// TIA Portal V16 export
// export: Created 2022-09-01T13:58:56.9257321Z, ExportSetting WithDefaults, DisplayName Totally Integrated Automation Portal, DisplayVersion V16, DisplayName TIA Portal Version Control Interface, DisplayVersion V16, DisplayName TIA Portal Openness, DisplayVersion V16, DisplayName STEP 7 Professional, DisplayVersion V16, DisplayName STEP 7 Safety, DisplayVersion V16, DisplayName WinCC Advanced, DisplayVersion V16
DATA_BLOCK "Inputs_HMI"   // DB6
{ S7_Optimized_Access := 'TRUE' }
VERSION : 0.1
// stored: AutoNumber true, IsOnlyStoredInLoadMemory false, IsRetainMemResEnabled false, IsWriteProtectedInAS false, MemoryReserve 100
   VAR RETAIN
      T_LAVAGEM : Time;
      T_RINSE : Time;
      T_STOP_BOMBAS : Time;
      T_POS_EVS : Time;
      ENABLE_CICLO_FILT1 : Bool;
      ENABLE_CICLO_FILT2 : Bool;
   END_VAR
   VAR
      START_CICLO_FILT1 : Bool;
      START_CICLO_FILT2 : Bool;
      STOP_CICLO : Bool;
      REARME : Bool;
      "MAN/AUTO" : Bool;
      "ON_OFF_EV1.1" : Bool;
      "ON_OFF_EV2.1" : Bool;
      "ON_OFF_EV3.1" : Bool;
      "ON_OFF_EV4.1" : Bool;
      "ON_OFF_EV5.1" : Bool;
      "ON_OFF_EV1.2" : Bool;
      "ON_OFF_EV2.2" : Bool;
      "ON_OFF_EV3.2" : Bool;
      "ON_OFF_EV4.2" : Bool;
      "ON_OFF_EV5.2" : Bool;
   END_VAR
   VAR RETAIN
      "MAN/AUTO_BOMBAS" : Bool;
      T_ALTERNANCIA_BOMBAS : Real;
   END_VAR
   VAR
      ON_OFF_BOMBA_1 : Bool;
      ON_OFF_BOMBA_2 : Bool;
      ON_OFF_BOMBA_3 : Bool;
      RESET_CNT_B1 : Bool;
      RESET_CNT_B2 : Bool;
      RESET_CNT_B3 : Bool;
   END_VAR
   VAR RETAIN
      SP_PRESS_FILT1 : Real;
      SP_PRESS_FILT2 : Real;
   END_VAR
BEGIN
END_DATA_BLOCK
